// ---- DUTs/IO/Boxes/EL3204_B6248F5B.TcDUT
{attribute 'GeneratedUsingTerminal: EL3204-0000-0017'}
{attribute addProperty BoxType "EL3204-0000-0017"}
{attribute addProperty Description "EL3204 4Ch. Ana. Input PT100 (RTD)"}
{attribute addProperty Physics "KK"}
{attribute addProperty Id "RTD_Inputs_Channel_1AT %I*AI_Standard_Channel_4A3944819RTD_Inputs_Channel_2AT %I*AI_Standard_Channel_4A3944819RTD_Inputs_Channel_3AT %I*AI_Standard_Channel_4A3944819RTD_Inputs_Channel_4AT %I*AI_Standard_Channel_4A3944819WcStateAT %I*WcState_9091E0EB2InfoDataAT %I*InfoData_32EB74EA10"}
{attribute addProperty CRC "3055849307"}
{attribute addProperty Size "48"}
TYPE EL3204_B6248F5B EXTENDS EtcSlaveTerminalBase_947E5A46 :
STRUCT
	{attribute addProperty Name "RTD_Inputs_Channel_1"}
	RTD_Inputs_Channel_1 : AI_Standard_Channel_4A394481;
	{attribute addProperty Name "RTD_Inputs_Channel_2"}
	RTD_Inputs_Channel_2 : AI_Standard_Channel_4A394481;
	{attribute addProperty Name "RTD_Inputs_Channel_3"}
	RTD_Inputs_Channel_3 : AI_Standard_Channel_4A394481;
	{attribute addProperty Name "RTD_Inputs_Channel_4"}
	RTD_Inputs_Channel_4 : AI_Standard_Channel_4A394481;
	{attribute addProperty Name "WcState"}
	WcState : WcState_9091E0EB;
	{attribute addProperty Name "InfoData"}
	InfoData : InfoData_32EB74EA;
END_STRUCT
END_TYPE

// ---- DUTs/IO/Boxes/EL3204_988CC224.TcDUT
{attribute 'GeneratedUsingTerminal: EL3204-0162-0016'}
{attribute addProperty BoxType "EL3204-0162-0016"}
{attribute addProperty Description "EL3204-0162 2Ch. Ana. In. PT100 (RTD), 2Ch. Ana. In. +/-10V, 0-10V configurable"}
{attribute addProperty Physics "KK"}
{attribute addProperty Id "RTD_Inputs_Channel_1AT %I*AI_Standard_Channel_4A3944819RTD_Inputs_Channel_2AT %I*AI_Standard_Channel_4A3944819AI_Standard_Channel_1AT %I*AI_Standard_Channel_4A3944819AI_Standard_Channel_2AT %I*AI_Standard_Channel_4A3944819WcStateAT %I*WcState_9091E0EB2InfoDataAT %I*InfoData_32EB74EA10"}
{attribute addProperty CRC "2559361572"}
{attribute addProperty Size "48"}
TYPE EL3204_988CC224 EXTENDS EtcSlaveTerminalBase_947E5A46 :
STRUCT
	{attribute addProperty Name "RTD_Inputs_Channel_1"}
	RTD_Inputs_Channel_1 : AI_Standard_Channel_4A394481;
	{attribute addProperty Name "RTD_Inputs_Channel_2"}
	RTD_Inputs_Channel_2 : AI_Standard_Channel_4A394481;
	{attribute addProperty Name "AI_Standard_Channel_1"}
	AI_Standard_Channel_1 : AI_Standard_Channel_4A394481;
	{attribute addProperty Name "AI_Standard_Channel_2"}
	AI_Standard_Channel_2 : AI_Standard_Channel_4A394481;
	{attribute addProperty Name "WcState"}
	WcState : WcState_9091E0EB;
	{attribute addProperty Name "InfoData"}
	InfoData : InfoData_32EB74EA;
END_STRUCT
END_TYPE

// ---- DUTs/IO/Boxes/EL3204_8BBE23EA.TcDUT
{attribute 'GeneratedUsingTerminal: EL3204-0200-0016'}
{attribute addProperty BoxType "EL3204-0200-0016"}
{attribute addProperty Description "EL3204-0200 4Ch. Ana. In. PT1000 (RTD)"}
{attribute addProperty Physics "KK"}
{attribute addProperty Id "RTD_Inputs_Channel_1AT %I*RTD_Inputs_Channel_9575FEA17RTD_Inputs_Channel_2AT %I*RTD_Inputs_Channel_9575FEA17RTD_Inputs_Channel_3AT %I*RTD_Inputs_Channel_9575FEA17RTD_Inputs_Channel_4AT %I*RTD_Inputs_Channel_9575FEA17WcStateAT %I*WcState_9091E0EB2InfoDataAT %I*InfoData_32EB74EA10"}
{attribute addProperty CRC "2344494058"}
{attribute addProperty Size "40"}
TYPE EL3204_8BBE23EA EXTENDS EtcSlaveTerminalBase_947E5A46 :
STRUCT
	{attribute addProperty Name "RTD_Inputs_Channel_1"}
	RTD_Inputs_Channel_1 : RTD_Inputs_Channel_9575FEA1;
	{attribute addProperty Name "RTD_Inputs_Channel_2"}
	RTD_Inputs_Channel_2 : RTD_Inputs_Channel_9575FEA1;
	{attribute addProperty Name "RTD_Inputs_Channel_3"}
	RTD_Inputs_Channel_3 : RTD_Inputs_Channel_9575FEA1;
	{attribute addProperty Name "RTD_Inputs_Channel_4"}
	RTD_Inputs_Channel_4 : RTD_Inputs_Channel_9575FEA1;
	{attribute addProperty Name "WcState"}
	WcState : WcState_9091E0EB;
	{attribute addProperty Name "InfoData"}
	InfoData : InfoData_32EB74EA;
END_STRUCT
END_TYPE

// ---- DUTs/IO/Boxes/EL3208_E885804F.TcDUT
{attribute 'GeneratedUsingTerminal: EL3208-0000-0017'}
{attribute addProperty BoxType "EL3208-0000-0017"}
{attribute addProperty Description "EL3208 8Ch. Ana. Input PT100 (RTD)"}
{attribute addProperty Physics "KK"}
{attribute addProperty Id "RTD_Inputs_Channel_1AT %I*RTD_Inputs_Channel_9575FEA17RTD_Inputs_Channel_2AT %I*RTD_Inputs_Channel_9575FEA17RTD_Inputs_Channel_3AT %I*RTD_Inputs_Channel_9575FEA17RTD_Inputs_Channel_4AT %I*RTD_Inputs_Channel_9575FEA17RTD_Inputs_Channel_5AT %I*RTD_Inputs_Channel_9575FEA17RTD_Inputs_Channel_6AT %I*RTD_Inputs_Channel_9575FEA17RTD_Inputs_Channel_7AT %I*RTD_Inputs_Channel_9575FEA17RTD_Inputs_Channel_8AT %I*RTD_Inputs_Channel_9575FEA17WcStateAT %I*WcState_9091E0EB2InfoDataAT %I*InfoData_32EB74EA10"}
{attribute addProperty CRC "3901063247"}
{attribute addProperty Size "68"}
TYPE EL3208_E885804F EXTENDS EtcSlaveTerminalBase_947E5A46 :
STRUCT
	{attribute addProperty Name "RTD_Inputs_Channel_1"}
	RTD_Inputs_Channel_1 : RTD_Inputs_Channel_9575FEA1;
	{attribute addProperty Name "RTD_Inputs_Channel_2"}
	RTD_Inputs_Channel_2 : RTD_Inputs_Channel_9575FEA1;
	{attribute addProperty Name "RTD_Inputs_Channel_3"}
	RTD_Inputs_Channel_3 : RTD_Inputs_Channel_9575FEA1;
	{attribute addProperty Name "RTD_Inputs_Channel_4"}
	RTD_Inputs_Channel_4 : RTD_Inputs_Channel_9575FEA1;
	{attribute addProperty Name "RTD_Inputs_Channel_5"}
	RTD_Inputs_Channel_5 : RTD_Inputs_Channel_9575FEA1;
	{attribute addProperty Name "RTD_Inputs_Channel_6"}
	RTD_Inputs_Channel_6 : RTD_Inputs_Channel_9575FEA1;
	{attribute addProperty Name "RTD_Inputs_Channel_7"}
	RTD_Inputs_Channel_7 : RTD_Inputs_Channel_9575FEA1;
	{attribute addProperty Name "RTD_Inputs_Channel_8"}
	RTD_Inputs_Channel_8 : RTD_Inputs_Channel_9575FEA1;
	{attribute addProperty Name "WcState"}
	WcState : WcState_9091E0EB;
	{attribute addProperty Name "InfoData"}
	InfoData : InfoData_32EB74EA;
END_STRUCT
END_TYPE

// ---- DUTs/IO/Boxes/EL3214_8BBE23EA.TcDUT
{attribute 'GeneratedUsingTerminal: EL3214-0000-0016'}
{attribute addProperty BoxType "EL3214-0000-0016"}
{attribute addProperty Description "EL3214 4Ch. Ana. Input PT100 (RTD)"}
{attribute addProperty Physics "KK"}
{attribute addProperty Id "RTD_Inputs_Channel_1AT %I*RTD_Inputs_Channel_9575FEA17RTD_Inputs_Channel_2AT %I*RTD_Inputs_Channel_9575FEA17RTD_Inputs_Channel_3AT %I*RTD_Inputs_Channel_9575FEA17RTD_Inputs_Channel_4AT %I*RTD_Inputs_Channel_9575FEA17WcStateAT %I*WcState_9091E0EB2InfoDataAT %I*InfoData_32EB74EA10"}
{attribute addProperty CRC "2344494058"}
{attribute addProperty Size "40"}
TYPE EL3214_8BBE23EA EXTENDS EtcSlaveTerminalBase_947E5A46 :
STRUCT
	{attribute addProperty Name "RTD_Inputs_Channel_1"}
	RTD_Inputs_Channel_1 : RTD_Inputs_Channel_9575FEA1;
	{attribute addProperty Name "RTD_Inputs_Channel_2"}
	RTD_Inputs_Channel_2 : RTD_Inputs_Channel_9575FEA1;
	{attribute addProperty Name "RTD_Inputs_Channel_3"}
	RTD_Inputs_Channel_3 : RTD_Inputs_Channel_9575FEA1;
	{attribute addProperty Name "RTD_Inputs_Channel_4"}
	RTD_Inputs_Channel_4 : RTD_Inputs_Channel_9575FEA1;
	{attribute addProperty Name "WcState"}
	WcState : WcState_9091E0EB;
	{attribute addProperty Name "InfoData"}
	InfoData : InfoData_32EB74EA;
END_STRUCT
END_TYPE

// ---- DUTs/IO/Boxes/EL3218_E885804F.TcDUT
{attribute 'GeneratedUsingTerminal: EL3218-0000-0016'}
{attribute addProperty BoxType "EL3218-0000-0016"}
{attribute addProperty Description "EL3218-0000 8Ch. Ana. Input PT100 (RTD)"}
{attribute addProperty Physics "KK"}
{attribute addProperty Id "RTD_Inputs_Channel_1AT %I*RTD_Inputs_Channel_9575FEA17RTD_Inputs_Channel_2AT %I*RTD_Inputs_Channel_9575FEA17RTD_Inputs_Channel_3AT %I*RTD_Inputs_Channel_9575FEA17RTD_Inputs_Channel_4AT %I*RTD_Inputs_Channel_9575FEA17RTD_Inputs_Channel_5AT %I*RTD_Inputs_Channel_9575FEA17RTD_Inputs_Channel_6AT %I*RTD_Inputs_Channel_9575FEA17RTD_Inputs_Channel_7AT %I*RTD_Inputs_Channel_9575FEA17RTD_Inputs_Channel_8AT %I*RTD_Inputs_Channel_9575FEA17WcStateAT %I*WcState_9091E0EB2InfoDataAT %I*InfoData_32EB74EA10"}
{attribute addProperty CRC "3901063247"}
{attribute addProperty Size "68"}
TYPE EL3218_E885804F EXTENDS EtcSlaveTerminalBase_947E5A46 :
STRUCT
	{attribute addProperty Name "RTD_Inputs_Channel_1"}
	RTD_Inputs_Channel_1 : RTD_Inputs_Channel_9575FEA1;
	{attribute addProperty Name "RTD_Inputs_Channel_2"}
	RTD_Inputs_Channel_2 : RTD_Inputs_Channel_9575FEA1;
	{attribute addProperty Name "RTD_Inputs_Channel_3"}
	RTD_Inputs_Channel_3 : RTD_Inputs_Channel_9575FEA1;
	{attribute addProperty Name "RTD_Inputs_Channel_4"}
	RTD_Inputs_Channel_4 : RTD_Inputs_Channel_9575FEA1;
	{attribute addProperty Name "RTD_Inputs_Channel_5"}
	RTD_Inputs_Channel_5 : RTD_Inputs_Channel_9575FEA1;
	{attribute addProperty Name "RTD_Inputs_Channel_6"}
	RTD_Inputs_Channel_6 : RTD_Inputs_Channel_9575FEA1;
	{attribute addProperty Name "RTD_Inputs_Channel_7"}
	RTD_Inputs_Channel_7 : RTD_Inputs_Channel_9575FEA1;
	{attribute addProperty Name "RTD_Inputs_Channel_8"}
	RTD_Inputs_Channel_8 : RTD_Inputs_Channel_9575FEA1;
	{attribute addProperty Name "WcState"}
	WcState : WcState_9091E0EB;
	{attribute addProperty Name "InfoData"}
	InfoData : InfoData_32EB74EA;
END_STRUCT
END_TYPE

// ---- DUTs/IO/Boxes/EL3255_70670831.TcDUT
{attribute 'GeneratedUsingTerminal: EL3255-0000-0016'}
{attribute addProperty BoxType "EL3255-0000-0016"}
{attribute addProperty Description "EL3255 5Ch. potentiometer measurement with sensor supply"}
{attribute addProperty Physics "KK"}
{attribute addProperty Id "RTD_Standard_Channel_1AT %I*RTD_Standard_Channel_A8DF64E310RTD_Standard_Channel_2AT %I*RTD_Standard_Channel_A8DF64E310RTD_Standard_Channel_3AT %I*RTD_Standard_Channel_A8DF64E310RTD_Standard_Channel_4AT %I*RTD_Standard_Channel_A8DF64E310RTD_Standard_Channel_5AT %I*RTD_Standard_Channel_A8DF64E310WcStateAT %I*WcState_9091E0EB2InfoDataAT %I*InfoData_32EB74EA10"}
{attribute addProperty CRC "1885800497"}
{attribute addProperty Size "62"}
TYPE EL3255_70670831 EXTENDS EtcSlaveTerminalBase_947E5A46 :
STRUCT
	{attribute addProperty Name "RTD_Standard_Channel_1"}
	RTD_Standard_Channel_1 : RTD_Standard_Channel_A8DF64E3;
	{attribute addProperty Name "RTD_Standard_Channel_2"}
	RTD_Standard_Channel_2 : RTD_Standard_Channel_A8DF64E3;
	{attribute addProperty Name "RTD_Standard_Channel_3"}
	RTD_Standard_Channel_3 : RTD_Standard_Channel_A8DF64E3;
	{attribute addProperty Name "RTD_Standard_Channel_4"}
	RTD_Standard_Channel_4 : RTD_Standard_Channel_A8DF64E3;
	{attribute addProperty Name "RTD_Standard_Channel_5"}
	RTD_Standard_Channel_5 : RTD_Standard_Channel_A8DF64E3;
	{attribute addProperty Name "WcState"}
	WcState : WcState_9091E0EB;
	{attribute addProperty Name "InfoData"}
	InfoData : InfoData_32EB74EA;
END_STRUCT
END_TYPE

// ---- DUTs/IO/Boxes/EL3255_1972F7C0.TcDUT
{attribute 'GeneratedUsingTerminal: EL3255-0000-0017'}
{attribute addProperty BoxType "EL3255-0000-0017"}
{attribute addProperty Description "EL3255 5Ch. potentiometer measurement with sensor supply"}
{attribute addProperty Physics "KK"}
{attribute addProperty Id "AI_Standard_Channel_1AT %I*AI_Standard_Channel_A8DF64E310AI_Standard_Channel_2AT %I*AI_Standard_Channel_A8DF64E310AI_Standard_Channel_3AT %I*AI_Standard_Channel_A8DF64E310AI_Standard_Channel_4AT %I*AI_Standard_Channel_A8DF64E310AI_Standard_Channel_5AT %I*AI_Standard_Channel_A8DF64E310WcStateAT %I*WcState_9091E0EB2InfoDataAT %I*InfoData_32EB74EA10"}
{attribute addProperty CRC "426964928"}
{attribute addProperty Size "62"}
TYPE EL3255_1972F7C0 EXTENDS EtcSlaveTerminalBase_947E5A46 :
STRUCT
	{attribute addProperty Name "AI_Standard_Channel_1"}
	AI_Standard_Channel_1 : AI_Standard_Channel_A8DF64E3;
	{attribute addProperty Name "AI_Standard_Channel_2"}
	AI_Standard_Channel_2 : AI_Standard_Channel_A8DF64E3;
	{attribute addProperty Name "AI_Standard_Channel_3"}
	AI_Standard_Channel_3 : AI_Standard_Channel_A8DF64E3;
	{attribute addProperty Name "AI_Standard_Channel_4"}
	AI_Standard_Channel_4 : AI_Standard_Channel_A8DF64E3;
	{attribute addProperty Name "AI_Standard_Channel_5"}
	AI_Standard_Channel_5 : AI_Standard_Channel_A8DF64E3;
	{attribute addProperty Name "WcState"}
	WcState : WcState_9091E0EB;
	{attribute addProperty Name "InfoData"}
	InfoData : InfoData_32EB74EA;
END_STRUCT
END_TYPE

// ---- DUTs/IO/Boxes/EL3255_B4D4BD51.TcDUT
{attribute 'GeneratedUsingTerminal: EL3255-0000-0020'}
{attribute addProperty BoxType "EL3255-0000-0020"}
{attribute addProperty Description "EL3255 5Ch. potentiometer measurement with sensor supply"}
{attribute addProperty Physics "KK"}
{attribute addProperty Id "AI_Compact_Channel_1AT %I*AI_Compact_Channel_80E77D6A2AI_Standard_Channel_3AT %I*AI_Standard_Channel_A8DF64E310AI_Standard_Channel_4AT %I*AI_Standard_Channel_A8DF64E310AI_Standard_Channel_5AT %I*AI_Standard_Channel_A8DF64E310WcStateAT %I*WcState_9091E0EB2InfoDataAT %I*InfoData_32EB74EA10"}
{attribute addProperty CRC "3033840977"}
{attribute addProperty Size "44"}
TYPE EL3255_B4D4BD51 EXTENDS EtcSlaveTerminalBase_947E5A46 :
STRUCT
	{attribute addProperty Name "AI_Compact_Channel_1"}
	AI_Compact_Channel_1 : AI_Compact_Channel_80E77D6A;
	{attribute addProperty Name "AI_Standard_Channel_3"}
	AI_Standard_Channel_3 : AI_Standard_Channel_A8DF64E3;
	{attribute addProperty Name "AI_Standard_Channel_4"}
	AI_Standard_Channel_4 : AI_Standard_Channel_A8DF64E3;
	{attribute addProperty Name "AI_Standard_Channel_5"}
	AI_Standard_Channel_5 : AI_Standard_Channel_A8DF64E3;
	{attribute addProperty Name "WcState"}
	WcState : WcState_9091E0EB;
	{attribute addProperty Name "InfoData"}
	InfoData : InfoData_32EB74EA;
END_STRUCT
END_TYPE

// ---- DUTs/IO/Boxes/EL3311_768B3E67.TcDUT
{attribute 'GeneratedUsingTerminal: EL3311-0000-0016'}
{attribute addProperty BoxType "EL3311-0000-0016"}
{attribute addProperty Description "EL3311 1Ch. Ana. Input Thermocouple (TC)"}
{attribute addProperty Physics "KK"}
{attribute addProperty Id "TC_InputsAT %I*TC_Inputs_EA9DF21E9WcStateAT %I*WcState_9091E0EB2InfoDataAT %I*InfoData_32EB74EA10"}
{attribute addProperty CRC "1988836967"}
{attribute addProperty Size "21"}
TYPE EL3311_768B3E67 EXTENDS EtcSlaveTerminalBase_947E5A46 :
STRUCT
	{attribute addProperty Name "TC_Inputs"}
	TC_Inputs : TC_Inputs_EA9DF21E;
	{attribute addProperty Name "WcState"}
	WcState : WcState_9091E0EB;
	{attribute addProperty Name "InfoData"}
	InfoData : InfoData_32EB74EA;
END_STRUCT
END_TYPE

// ---- DUTs/IO/Boxes/EL3311_18A81F50.TcDUT
{attribute 'GeneratedUsingTerminal: EL3311-0000-0018'}
{attribute addProperty BoxType "EL3311-0000-0018"}
{attribute addProperty Description "EL3311 1Ch. Ana. Input Thermocouple (TC)"}
{attribute addProperty Physics "KK"}
{attribute addProperty Id "TC_InputsAT %I*AI_Standard_Channel_4A3944819WcStateAT %I*WcState_9091E0EB2InfoDataAT %I*InfoData_32EB74EA10"}
{attribute addProperty CRC "413671248"}
{attribute addProperty Size "21"}
TYPE EL3311_18A81F50 EXTENDS EtcSlaveTerminalBase_947E5A46 :
STRUCT
	{attribute addProperty Name "TC_Inputs"}
	TC_Inputs : AI_Standard_Channel_4A394481;
	{attribute addProperty Name "WcState"}
	WcState : WcState_9091E0EB;
	{attribute addProperty Name "InfoData"}
	InfoData : InfoData_32EB74EA;
END_STRUCT
END_TYPE

// ---- DUTs/IO/Boxes/EL3312_48655483.TcDUT
{attribute 'GeneratedUsingTerminal: EL3312-0000-0016'}
{attribute addProperty BoxType "EL3312-0000-0016"}
{attribute addProperty Description "EL3312 2Ch. Ana. Input Thermocouple (TC)"}
{attribute addProperty Physics "KK"}
{attribute addProperty Id "TC_Inputs_Channel_1AT %I*TC_Inputs_Channel_EA9DF21E9TC_Inputs_Channel_2AT %I*TC_Inputs_Channel_EA9DF21E9WcStateAT %I*WcState_9091E0EB2InfoDataAT %I*InfoData_32EB74EA10"}
{attribute addProperty CRC "1214600323"}
{attribute addProperty Size "30"}
TYPE EL3312_48655483 EXTENDS EtcSlaveTerminalBase_947E5A46 :
STRUCT
	{attribute addProperty Name "TC_Inputs_Channel_1"}
	TC_Inputs_Channel_1 : TC_Inputs_Channel_EA9DF21E;
	{attribute addProperty Name "TC_Inputs_Channel_2"}
	TC_Inputs_Channel_2 : TC_Inputs_Channel_EA9DF21E;
	{attribute addProperty Name "WcState"}
	WcState : WcState_9091E0EB;
	{attribute addProperty Name "InfoData"}
	InfoData : InfoData_32EB74EA;
END_STRUCT
END_TYPE

// ---- DUTs/IO/Boxes/EL3312_BE98AB26.TcDUT
{attribute 'GeneratedUsingTerminal: EL3312-0000-0018'}
{attribute addProperty BoxType "EL3312-0000-0018"}
{attribute addProperty Description "EL3312 2Ch. Ana. Input Thermocouple (TC)"}
{attribute addProperty Physics "KK"}
{attribute addProperty Id "TC_Inputs_Channel_1AT %I*AI_Standard_Channel_4A3944819TC_Inputs_Channel_2AT %I*AI_Standard_Channel_4A3944819WcStateAT %I*WcState_9091E0EB2InfoDataAT %I*InfoData_32EB74EA10"}
{attribute addProperty CRC "3197676326"}
{attribute addProperty Size "30"}
TYPE EL3312_BE98AB26 EXTENDS EtcSlaveTerminalBase_947E5A46 :
STRUCT
	{attribute addProperty Name "TC_Inputs_Channel_1"}
	TC_Inputs_Channel_1 : AI_Standard_Channel_4A394481;
	{attribute addProperty Name "TC_Inputs_Channel_2"}
	TC_Inputs_Channel_2 : AI_Standard_Channel_4A394481;
	{attribute addProperty Name "WcState"}
	WcState : WcState_9091E0EB;
	{attribute addProperty Name "InfoData"}
	InfoData : InfoData_32EB74EA;
END_STRUCT
END_TYPE

// ---- DUTs/IO/Boxes/EL3314_18BBAF47.TcDUT
{attribute 'GeneratedUsingTerminal: EL3314-0000-0016'}
{attribute addProperty BoxType "EL3314-0000-0016"}
{attribute addProperty Description "EL3314 4Ch. Ana. Input Thermocouple (TC)"}
{attribute addProperty Physics "KK"}
{attribute addProperty Id "TC_Inputs_Channel_1AT %I*TC_Inputs_Channel_EA9DF21E9TC_Inputs_Channel_2AT %I*TC_Inputs_Channel_EA9DF21E9TC_Inputs_Channel_3AT %I*TC_Inputs_Channel_EA9DF21E9TC_Inputs_Channel_4AT %I*TC_Inputs_Channel_EA9DF21E9WcStateAT %I*WcState_9091E0EB2InfoDataAT %I*InfoData_32EB74EA10"}
{attribute addProperty CRC "414953287"}
{attribute addProperty Size "48"}
TYPE EL3314_18BBAF47 EXTENDS EtcSlaveTerminalBase_947E5A46 :
STRUCT
	{attribute addProperty Name "TC_Inputs_Channel_1"}
	TC_Inputs_Channel_1 : TC_Inputs_Channel_EA9DF21E;
	{attribute addProperty Name "TC_Inputs_Channel_2"}
	TC_Inputs_Channel_2 : TC_Inputs_Channel_EA9DF21E;
	{attribute addProperty Name "TC_Inputs_Channel_3"}
	TC_Inputs_Channel_3 : TC_Inputs_Channel_EA9DF21E;
	{attribute addProperty Name "TC_Inputs_Channel_4"}
	TC_Inputs_Channel_4 : TC_Inputs_Channel_EA9DF21E;
	{attribute addProperty Name "WcState"}
	WcState : WcState_9091E0EB;
	{attribute addProperty Name "InfoData"}
	InfoData : InfoData_32EB74EA;
END_STRUCT
END_TYPE

// ---- DUTs/IO/Boxes/EL3314_E65CDB1C.TcDUT
{attribute 'GeneratedUsingTerminal: EL3314-0000-0018'}
{attribute addProperty BoxType "EL3314-0000-0018"}
{attribute addProperty Description "EL3314 4Ch. Ana. Input Thermocouple (TC)"}
{attribute addProperty Physics "KK"}
{attribute addProperty Id "TC_Inputs_Channel_1AT %I*AI_Standard_Channel_4A3944819TC_Inputs_Channel_2AT %I*AI_Standard_Channel_4A3944819TC_Inputs_Channel_3AT %I*AI_Standard_Channel_4A3944819TC_Inputs_Channel_4AT %I*AI_Standard_Channel_4A3944819WcStateAT %I*WcState_9091E0EB2InfoDataAT %I*InfoData_32EB74EA10"}
{attribute addProperty CRC "3864845084"}
{attribute addProperty Size "48"}
TYPE EL3314_E65CDB1C EXTENDS EtcSlaveTerminalBase_947E5A46 :
STRUCT
	{attribute addProperty Name "TC_Inputs_Channel_1"}
	TC_Inputs_Channel_1 : AI_Standard_Channel_4A394481;
	{attribute addProperty Name "TC_Inputs_Channel_2"}
	TC_Inputs_Channel_2 : AI_Standard_Channel_4A394481;
	{attribute addProperty Name "TC_Inputs_Channel_3"}
	TC_Inputs_Channel_3 : AI_Standard_Channel_4A394481;
	{attribute addProperty Name "TC_Inputs_Channel_4"}
	TC_Inputs_Channel_4 : AI_Standard_Channel_4A394481;
	{attribute addProperty Name "WcState"}
	WcState : WcState_9091E0EB;
	{attribute addProperty Name "InfoData"}
	InfoData : InfoData_32EB74EA;
END_STRUCT
END_TYPE

// ---- DUTs/IO/Boxes/EL3314_6E4DFFE5.TcDUT
{attribute 'GeneratedUsingTerminal: EL3314-0002-0016'}
{attribute addProperty BoxType "EL3314-0002-0016"}
{attribute addProperty Description "EL3314-0002 4Ch. Ana Input Thermocouple (TC), Isolated Channels"}
{attribute addProperty Physics "KK"}
{attribute addProperty Id "TC_Inputs_Channel_1AT %I*TC_Inputs_Channel_4521310411TC_Inputs_Channel_2AT %I*TC_Inputs_Channel_4521310411TC_Inputs_Channel_3AT %I*TC_Inputs_Channel_4521310411TC_Inputs_Channel_4AT %I*TC_Inputs_Channel_4521310411WcStateAT %I*WcState_9091E0EB2InfoDataAT %I*InfoData_32EB74EA10"}
{attribute addProperty CRC "1850605541"}
{attribute addProperty Size "56"}
TYPE EL3314_6E4DFFE5 EXTENDS EtcSlaveTerminalBase_947E5A46 :
STRUCT
	{attribute addProperty Name "TC_Inputs_Channel_1"}
	TC_Inputs_Channel_1 : TC_Inputs_Channel_45213104;
	{attribute addProperty Name "TC_Inputs_Channel_2"}
	TC_Inputs_Channel_2 : TC_Inputs_Channel_45213104;
	{attribute addProperty Name "TC_Inputs_Channel_3"}
	TC_Inputs_Channel_3 : TC_Inputs_Channel_45213104;
	{attribute addProperty Name "TC_Inputs_Channel_4"}
	TC_Inputs_Channel_4 : TC_Inputs_Channel_45213104;
	{attribute addProperty Name "WcState"}
	WcState : WcState_9091E0EB;
	{attribute addProperty Name "InfoData"}
	InfoData : InfoData_32EB74EA;
END_STRUCT
END_TYPE

// ---- DUTs/IO/Boxes/EL3318_44C149FC.TcDUT
{attribute 'GeneratedUsingTerminal: EL3318-0000-0016'}
{attribute addProperty BoxType "EL3318-0000-0016"}
{attribute addProperty Description "EL3318 8Ch. Ana Input Thermocouple (TC)"}
{attribute addProperty Physics "KK"}
{attribute addProperty Id "TC_Channel_1AT %I*TC_Channel_9575FEA17TC_Channel_2AT %I*TC_Channel_9575FEA17TC_Channel_3AT %I*TC_Channel_9575FEA17TC_Channel_4AT %I*TC_Channel_9575FEA17TC_Channel_5AT %I*TC_Channel_9575FEA17TC_Channel_6AT %I*TC_Channel_9575FEA17TC_Channel_7AT %I*TC_Channel_9575FEA17TC_Channel_8AT %I*TC_Channel_9575FEA17WcStateAT %I*WcState_9091E0EB2InfoDataAT %I*InfoData_32EB74EA10"}
{attribute addProperty CRC "1153518076"}
{attribute addProperty Size "68"}
TYPE EL3318_44C149FC EXTENDS EtcSlaveTerminalBase_947E5A46 :
STRUCT
	{attribute addProperty Name "TC_Channel_1"}
	TC_Channel_1 : TC_Channel_9575FEA1;
	{attribute addProperty Name "TC_Channel_2"}
	TC_Channel_2 : TC_Channel_9575FEA1;
	{attribute addProperty Name "TC_Channel_3"}
	TC_Channel_3 : TC_Channel_9575FEA1;
	{attribute addProperty Name "TC_Channel_4"}
	TC_Channel_4 : TC_Channel_9575FEA1;
	{attribute addProperty Name "TC_Channel_5"}
	TC_Channel_5 : TC_Channel_9575FEA1;
	{attribute addProperty Name "TC_Channel_6"}
	TC_Channel_6 : TC_Channel_9575FEA1;
	{attribute addProperty Name "TC_Channel_7"}
	TC_Channel_7 : TC_Channel_9575FEA1;
	{attribute addProperty Name "TC_Channel_8"}
	TC_Channel_8 : TC_Channel_9575FEA1;
	{attribute addProperty Name "WcState"}
	WcState : WcState_9091E0EB;
	{attribute addProperty Name "InfoData"}
	InfoData : InfoData_32EB74EA;
END_STRUCT
END_TYPE

// ---- DUTs/IO/Boxes/EL3351_6847F283.TcDUT
{attribute 'GeneratedUsingTerminal: EL3351-0000-0016'}
{attribute addProperty BoxType "EL3351-0000-0016"}
{attribute addProperty Description "EL3351 1Ch. Ana. Input Resistor Bridge Terminal, Diff. 16bit "}
{attribute addProperty Physics "KK"}
{attribute addProperty Id "AIBridge_InputsAT %I*AIBridge_Inputs_555AA1E89AISupply_InputsAT %I*AISupply_Inputs_555AA1E89WcStateAT %I*WcState_9091E0EB2InfoDataAT %I*InfoData_32EB74EA10"}
{attribute addProperty CRC "1749545603"}
{attribute addProperty Size "30"}
TYPE EL3351_6847F283 EXTENDS EtcSlaveTerminalBase_947E5A46 :
STRUCT
	{attribute addProperty Name "AIBridge_Inputs"}
	AIBridge_Inputs : AIBridge_Inputs_555AA1E8;
	{attribute addProperty Name "AISupply_Inputs"}
	AISupply_Inputs : AISupply_Inputs_555AA1E8;
	{attribute addProperty Name "WcState"}
	WcState : WcState_9091E0EB;
	{attribute addProperty Name "InfoData"}
	InfoData : InfoData_32EB74EA;
END_STRUCT
END_TYPE

// ---- DUTs/IO/Boxes/EL3356_8E3EBEA0.TcDUT
{attribute 'GeneratedUsingTerminal: EL3356-0000-0017'}
{attribute addProperty BoxType "EL3356-0000-0017"}
{attribute addProperty Description "EL3356 1Ch. Ana. Input Resistor Bridge Terminal, 16bit, High Precision"}
{attribute addProperty Physics "KK"}
{attribute addProperty Id "RMB_StatusAT %I*RMB_Status_C0E100AA7RMB_Value_INT32AT %I*RMB_Value_INT_E9189C4B4RMB_ControlAT %Q*RMB_Control_4997AEF64WcStateAT %I*WcState_9091E0EB2InfoDataAT %I*InfoData_32EB74EA10"}
{attribute addProperty CRC "2386476704"}
{attribute addProperty Size "27"}
TYPE EL3356_8E3EBEA0 EXTENDS EtcSlaveTerminalBase_947E5A46 :
STRUCT
	{attribute addProperty Name "RMB_Status"}
	RMB_Status : RMB_Status_C0E100AA;
	{attribute addProperty Name "RMB_Value_INT32"}
	RMB_Value_INT32 : RMB_Value_INT_E9189C4B;
	{attribute addProperty Name "RMB_Control"}
	RMB_Control : RMB_Control_4997AEF6;
	{attribute addProperty Name "WcState"}
	WcState : WcState_9091E0EB;
	{attribute addProperty Name "InfoData"}
	InfoData : InfoData_32EB74EA;
END_STRUCT
END_TYPE

// ---- DUTs/IO/Boxes/EL3403_A37C91B8.TcDUT
{attribute 'GeneratedUsingTerminal: EL3403-0000-0017'}
{attribute addProperty BoxType "EL3403-0000-0017"}
{attribute addProperty Description "EL3403 3Ch. Power Measuring"}
{attribute addProperty Physics "KK"}
{attribute addProperty Id "PM_Inputs_Channel_1AT %I*PM_Inputs_Channel_6909D40619PM_Inputs_Channel_2AT %I*PM_Inputs_Channel_6909D40619PM_Inputs_Channel_3AT %I*PM_Inputs_Channel_6909D40619PM_Status_dataAT %I*PM_Status_data_0FD072A05PM_Outputs_Channel_1AT %Q*PM_Outputs_Channel_E5FBDE301PM_Outputs_Channel_2AT %Q*PM_Outputs_Channel_E5FBDE301PM_Outputs_Channel_3AT %Q*PM_Outputs_Channel_E5FBDE301WcStateAT %I*WcState_9091E0EB2InfoDataAT %I*InfoData_32EB74EA10"}
{attribute addProperty CRC "2742849976"}
{attribute addProperty Size "77"}
TYPE EL3403_A37C91B8 EXTENDS EtcSlaveTerminalBase_947E5A46 :
STRUCT
	{attribute addProperty Name "PM_Inputs_Channel_1"}
	PM_Inputs_Channel_1 : PM_Inputs_Channel_6909D406;
	{attribute addProperty Name "PM_Inputs_Channel_2"}
	PM_Inputs_Channel_2 : PM_Inputs_Channel_6909D406;
	{attribute addProperty Name "PM_Inputs_Channel_3"}
	PM_Inputs_Channel_3 : PM_Inputs_Channel_6909D406;
	{attribute addProperty Name "PM_Status_data"}
	PM_Status_data : PM_Status_data_0FD072A0;
	{attribute addProperty Name "PM_Outputs_Channel_1"}
	PM_Outputs_Channel_1 : PM_Outputs_Channel_E5FBDE30;
	{attribute addProperty Name "PM_Outputs_Channel_2"}
	PM_Outputs_Channel_2 : PM_Outputs_Channel_E5FBDE30;
	{attribute addProperty Name "PM_Outputs_Channel_3"}
	PM_Outputs_Channel_3 : PM_Outputs_Channel_E5FBDE30;
	{attribute addProperty Name "WcState"}
	WcState : WcState_9091E0EB;
	{attribute addProperty Name "InfoData"}
	InfoData : InfoData_32EB74EA;
END_STRUCT
END_TYPE

// ---- DUTs/IO/Boxes/EL3403_B537021B.TcDUT
{attribute 'GeneratedUsingTerminal: EL3403-0000-0018'}
{attribute addProperty BoxType "EL3403-0000-0018"}
{attribute addProperty Description "EL3403 3Ch. Power Measuring"}
{attribute addProperty Physics "KK"}
{attribute addProperty Id "PM_Inputs_Channel_1AT %I*PM_Inputs_Channel_2468BF1D19PM_Inputs_Channel_2AT %I*PM_Inputs_Channel_2468BF1D19PM_Inputs_Channel_3AT %I*PM_Inputs_Channel_2468BF1D19PM_Status_dataAT %I*PM_Status_data_0FD072A05PM_Outputs_Channel_1AT %Q*PM_Outputs_Channel_E5FBDE301PM_Outputs_Channel_2AT %Q*PM_Outputs_Channel_E5FBDE301PM_Outputs_Channel_3AT %Q*PM_Outputs_Channel_E5FBDE301WcStateAT %I*WcState_9091E0EB2InfoDataAT %I*InfoData_32EB74EA10"}
{attribute addProperty CRC "3040281115"}
{attribute addProperty Size "77"}
TYPE EL3403_B537021B EXTENDS EtcSlaveTerminalBase_947E5A46 :
STRUCT
	{attribute addProperty Name "PM_Inputs_Channel_1"}
	PM_Inputs_Channel_1 : PM_Inputs_Channel_2468BF1D;
	{attribute addProperty Name "PM_Inputs_Channel_2"}
	PM_Inputs_Channel_2 : PM_Inputs_Channel_2468BF1D;
	{attribute addProperty Name "PM_Inputs_Channel_3"}
	PM_Inputs_Channel_3 : PM_Inputs_Channel_2468BF1D;
	{attribute addProperty Name "PM_Status_data"}
	PM_Status_data : PM_Status_data_0FD072A0;
	{attribute addProperty Name "PM_Outputs_Channel_1"}
	PM_Outputs_Channel_1 : PM_Outputs_Channel_E5FBDE30;
	{attribute addProperty Name "PM_Outputs_Channel_2"}
	PM_Outputs_Channel_2 : PM_Outputs_Channel_E5FBDE30;
	{attribute addProperty Name "PM_Outputs_Channel_3"}
	PM_Outputs_Channel_3 : PM_Outputs_Channel_E5FBDE30;
	{attribute addProperty Name "WcState"}
	WcState : WcState_9091E0EB;
	{attribute addProperty Name "InfoData"}
	InfoData : InfoData_32EB74EA;
END_STRUCT
END_TYPE

// ---- DUTs/IO/Boxes/EL3403_200C4240.TcDUT
{attribute 'GeneratedUsingTerminal: EL3403-0000-0022'}
{attribute addProperty BoxType "EL3403-0000-0022"}
{attribute addProperty Description "EL3403 3Ch. Power Measuring"}
{attribute addProperty Physics "KK"}
{attribute addProperty Id "PM_Inputs_Channel_1AT %I*PM_Inputs_Channel_2F86808618PM_Inputs_Channel_2AT %I*PM_Inputs_Channel_2F86808618PM_Inputs_Channel_3AT %I*PM_Inputs_Channel_2F86808618PM_Status_dataAT %I*PM_Status_data_2A9514CB4PM_Outputs_Channel_1AT %Q*PM_Outputs_Channel_E5FBDE301PM_Outputs_Channel_2AT %Q*PM_Outputs_Channel_E5FBDE301PM_Outputs_Channel_3AT %Q*PM_Outputs_Channel_E5FBDE301WcStateAT %I*WcState_9091E0EB2InfoDataAT %I*InfoData_32EB74EA10"}
{attribute addProperty CRC "537674304"}
{attribute addProperty Size "73"}
TYPE EL3403_200C4240 EXTENDS EtcSlaveTerminalBase_947E5A46 :
STRUCT
	{attribute addProperty Name "PM_Inputs_Channel_1"}
	PM_Inputs_Channel_1 : PM_Inputs_Channel_2F868086;
	{attribute addProperty Name "PM_Inputs_Channel_2"}
	PM_Inputs_Channel_2 : PM_Inputs_Channel_2F868086;
	{attribute addProperty Name "PM_Inputs_Channel_3"}
	PM_Inputs_Channel_3 : PM_Inputs_Channel_2F868086;
	{attribute addProperty Name "PM_Status_data"}
	PM_Status_data : PM_Status_data_2A9514CB;
	{attribute addProperty Name "PM_Outputs_Channel_1"}
	PM_Outputs_Channel_1 : PM_Outputs_Channel_E5FBDE30;
	{attribute addProperty Name "PM_Outputs_Channel_2"}
	PM_Outputs_Channel_2 : PM_Outputs_Channel_E5FBDE30;
	{attribute addProperty Name "PM_Outputs_Channel_3"}
	PM_Outputs_Channel_3 : PM_Outputs_Channel_E5FBDE30;
	{attribute addProperty Name "WcState"}
	WcState : WcState_9091E0EB;
	{attribute addProperty Name "InfoData"}
	InfoData : InfoData_32EB74EA;
END_STRUCT
END_TYPE

// ---- DUTs/IO/Boxes/EL3413_0563D894.TcDUT
{attribute 'GeneratedUsingTerminal: EL3413-0000-0016'}
{attribute addProperty BoxType "EL3413-0000-0016"}
{attribute addProperty Description "EL3413 3Ch. Power Measuring"}
{attribute addProperty Physics "KK"}
{attribute addProperty Id "PM_Inputs_Channel_1AT %I*PM_Inputs_Channel_345EAE5425PM_Inputs_Channel_2AT %I*PM_Inputs_Channel_345EAE5425PM_Inputs_Channel_3AT %I*PM_Inputs_Channel_345EAE5425PM_Inputs_AuxiliaryAT %I*PM_Inputs_Auxiliary_392D510B7PM_Outputs_Channel_1AT %Q*PM_Outputs_Channel_E5FBDE301PM_Outputs_Channel_2AT %Q*PM_Outputs_Channel_E5FBDE301PM_Outputs_Channel_3AT %Q*PM_Outputs_Channel_E5FBDE301PM_Outputs_AuxiliaryAT %Q*PM_Outputs_Auxiliary_6BC1946F2WcStateAT %I*WcState_9091E0EB2InfoDataAT %I*InfoData_32EB74EA10"}
{attribute addProperty CRC "90429588"}
{attribute addProperty Size "99"}
TYPE EL3413_0563D894 EXTENDS EtcSlaveTerminalBase_947E5A46 :
STRUCT
	{attribute addProperty Name "PM_Inputs_Channel_1"}
	PM_Inputs_Channel_1 : PM_Inputs_Channel_345EAE54;
	{attribute addProperty Name "PM_Inputs_Channel_2"}
	PM_Inputs_Channel_2 : PM_Inputs_Channel_345EAE54;
	{attribute addProperty Name "PM_Inputs_Channel_3"}
	PM_Inputs_Channel_3 : PM_Inputs_Channel_345EAE54;
	{attribute addProperty Name "PM_Inputs_Auxiliary"}
	PM_Inputs_Auxiliary : PM_Inputs_Auxiliary_392D510B;
	{attribute addProperty Name "PM_Outputs_Channel_1"}
	PM_Outputs_Channel_1 : PM_Outputs_Channel_E5FBDE30;
	{attribute addProperty Name "PM_Outputs_Channel_2"}
	PM_Outputs_Channel_2 : PM_Outputs_Channel_E5FBDE30;
	{attribute addProperty Name "PM_Outputs_Channel_3"}
	PM_Outputs_Channel_3 : PM_Outputs_Channel_E5FBDE30;
	{attribute addProperty Name "PM_Outputs_Auxiliary"}
	PM_Outputs_Auxiliary : PM_Outputs_Auxiliary_6BC1946F;
	{attribute addProperty Name "WcState"}
	WcState : WcState_9091E0EB;
	{attribute addProperty Name "InfoData"}
	InfoData : InfoData_32EB74EA;
END_STRUCT
END_TYPE

// ---- DUTs/IO/Boxes/EL3413_0EB67A0F.TcDUT
{attribute 'GeneratedUsingTerminal: EL3413-0000-0019'}
{attribute addProperty BoxType "EL3413-0000-0019"}
{attribute addProperty Description "EL3413 3Ch. Power Measuring"}
{attribute addProperty Physics "KK"}
{attribute addProperty Id "PM_Inputs_Channel_1AT %I*PM_Inputs_Channel_345EAE5425PM_Inputs_Channel_2AT %I*PM_Inputs_Channel_345EAE5425PM_Inputs_Channel_3AT %I*PM_Inputs_Channel_345EAE5425PM_Inputs_AuxiliaryAT %I*PM_Inputs_Auxiliary_3661DB6D9PM_Outputs_Channel_1AT %Q*PM_Outputs_Channel_E5FBDE301PM_Outputs_Channel_2AT %Q*PM_Outputs_Channel_E5FBDE301PM_Outputs_Channel_3AT %Q*PM_Outputs_Channel_E5FBDE301PM_Outputs_AuxiliaryAT %Q*PM_Outputs_Auxiliary_6BC1946F2WcStateAT %I*WcState_9091E0EB2InfoDataAT %I*InfoData_32EB74EA10"}
{attribute addProperty CRC "246839823"}
{attribute addProperty Size "101"}
TYPE EL3413_0EB67A0F EXTENDS EtcSlaveTerminalBase_947E5A46 :
STRUCT
	{attribute addProperty Name "PM_Inputs_Channel_1"}
	PM_Inputs_Channel_1 : PM_Inputs_Channel_345EAE54;
	{attribute addProperty Name "PM_Inputs_Channel_2"}
	PM_Inputs_Channel_2 : PM_Inputs_Channel_345EAE54;
	{attribute addProperty Name "PM_Inputs_Channel_3"}
	PM_Inputs_Channel_3 : PM_Inputs_Channel_345EAE54;
	{attribute addProperty Name "PM_Inputs_Auxiliary"}
	PM_Inputs_Auxiliary : PM_Inputs_Auxiliary_3661DB6D;
	{attribute addProperty Name "PM_Outputs_Channel_1"}
	PM_Outputs_Channel_1 : PM_Outputs_Channel_E5FBDE30;
	{attribute addProperty Name "PM_Outputs_Channel_2"}
	PM_Outputs_Channel_2 : PM_Outputs_Channel_E5FBDE30;
	{attribute addProperty Name "PM_Outputs_Channel_3"}
	PM_Outputs_Channel_3 : PM_Outputs_Channel_E5FBDE30;
	{attribute addProperty Name "PM_Outputs_Auxiliary"}
	PM_Outputs_Auxiliary : PM_Outputs_Auxiliary_6BC1946F;
	{attribute addProperty Name "WcState"}
	WcState : WcState_9091E0EB;
	{attribute addProperty Name "InfoData"}
	InfoData : InfoData_32EB74EA;
END_STRUCT
END_TYPE

// ---- DUTs/IO/Base/EtcSlaveBase_82538BE2.TcDUT

TYPE EtcSlaveBase_82538BE2 :
STRUCT
END_STRUCT
END_TYPE

// ---- DUTs/IO/Base/EtcSlaveBase_82538BE2.TcDUT

TYPE EtcSlaveBase_82538BE2 :
STRUCT
END_STRUCT
END_TYPE

// ---- DUTs/IO/Base/EtcSlaveBase_82538BE2.TcDUT

TYPE EtcSlaveBase_82538BE2 :
STRUCT
END_STRUCT
END_TYPE

// ---- DUTs/IO/Base/EtcSlaveTerminalBase_947E5A46.TcDUT

{attribute clr[Container(Layout.Stack)]}
{attribute clr[Group(Layout.GroupBox)]}
{attribute addProperty PreviousPort "Unknown"}
TYPE EtcSlaveTerminalBase_947E5A46 EXTENDS EtcSlaveBase_82538BE2 :
STRUCT
END_STRUCT
END_TYPE

// ---- DUTs/IO/Base/EtcSlaveBoxBase_77A0E4A7.TcDUT

{attribute clr[Container(Layout.Stack)]}
{attribute clr[Group(Layout.GroupBox)]}
{attribute addProperty PreviousPort "Unknown"}
TYPE EtcSlaveBoxBase_77A0E4A7 EXTENDS EtcSlaveBase_82538BE2 :
STRUCT
END_STRUCT
END_TYPE

// ---- DUTs/IO/Base/EtcSlaveEndTerminalBase_866C7F0C.TcDUT

{attribute clr[Container(Layout.Stack)]}
{attribute clr[Group(Layout.GroupBox)]}
{attribute addProperty PreviousPort "Unknown"}
TYPE EtcSlaveEndTerminalBase_866C7F0C EXTENDS EtcSlaveBase_82538BE2 :
STRUCT
END_STRUCT
END_TYPE

// ---- DUTs/IO/Base/InputBase_8311D824.TcDUT

TYPE InputBase_8311D824 :
STRUCT
END_STRUCT
END_TYPE

// ---- DUTs/IO/Base/OutputBase_10CEE7DE.TcDUT

TYPE OutputBase_10CEE7DE :
STRUCT
END_STRUCT
END_TYPE

// ---- DUTs/IO/Base/EtcMasterBase_62654B43.TcDUT

TYPE EtcMasterBase_62654B43 :
STRUCT
END_STRUCT
END_TYPE

// ---- GVLs/GVL_iXlinker.TcGVL
{attribute 'qualified_only'}
VAR_GLOBAL
		EtherCAT_Master_ELxxxx : EtherCAT_Master_ELxxxx_D0BA48C6;
END_VAR

// ---- POUs/MAIN.TcPOU
PROGRAM MAIN
VAR
END_VAR

END_PROGRAM
